Staubli VAL3: GeometryRS.dtx

public bool bIsScara = true
public bool bLinear = true
public bool bUseUserCenter
public bool bUseUserLimit = true
public num nSyncDist = 1
public num nWinDownStream
public num nWinUpStream
pointRs pVision[3]
  [0] = {x=392.598601, y=461.346273, z=-82.976862, rx=-180, ry=0, rz=55.644672, shoulder=righty, fatherId=world[0]}
  [1] = {x=445.324397, y=461.358462, z=-83.544881, rx=-180, ry=0, rz=55.723805, shoulder=righty, fatherId=world[0]}
  [2] = {x=392.992535, y=526.330074, z=-82.748547, rx=-180, ry=0, rz=55.461702, shoulder=righty, fatherId=world[0]}
pointRs pWinCenter = {fatherId=world[0]}
pointRs pWinDown[2]
  [0] = {x=671.469625, y=326.943975, z=-82.28712, rx=-180, ry=0, rz=88.395346, shoulder=righty, fatherId=world[0]}
  [1] = {x=483.971855, y=594.549314, z=-82.015497, rx=-180, ry=0, rz=65.421383, shoulder=righty, fatherId=world[0]}
pointRs pWinMiddle = {fatherId=world[0]}
pointRs pWinUp[2]
  [0] = {x=365.904087, y=326.91934, z=-82.602337, rx=-180, ry=0, rz=58.048606, shoulder=righty, fatherId=world[0]}
  [1] = {x=178.226561, y=594.767162, z=-82.846719, rx=-180, ry=0, rz=32.693909, shoulder=righty, fatherId=world[0]}
tool pointer = {z=100, fatherId=flange[0], ioLink=valve1}
